{attribute 'GeneratedUsingTerminal: KL6821'}
{attribute addProperty BoxType "KL6821"}
{attribute addProperty Id "Channel_1AT %Q*Channel_A4B48F2D0"}
{attribute addProperty CRC "4152132306"}
{attribute addProperty Size "0"}
TYPE KL6821_F77C82D2 :
STRUCT
	{attribute addProperty Name "Channel_1"}
	Channel_1 : Channel_A4B48F2D;
END_STRUCT
END_TYPE

(* stored: Version 1.2.0.0, ProductVersion 3.1.4024.9
   DUT KL6821_F77C82D2: Id {6fd7804e-a2fa-44af-8157-5cdd3353b9f0} *)
